FUNCTION_BLOCK FB_FBD_IL_LD_SamplePOU
VAR_INPUT
//	eOperation	: INT;
	eOperation	: E_Operation;
END_VAR
VAR_OUTPUT
	iResultC	: DINT;
END_VAR
VAR
	arrDataA	: ARRAY [1..iMax] OF DINT;
	arrDataB	: ARRAY [1..iMax] OF DINT;
	arrDataC	: ARRAY [1..iMax] OF DINT;
	I 			: DINT;
	bInit		: BOOL := TRUE;
	bEnd		: BOOL;
	bRepeat		: BOOL;
	bAtTheEnd	: BOOL;
END_VAR
VAR CONSTANT
	iMax 		: DINT := 10;
END_VAR
VAR // added by the converter: edge detectors and wires of the graphical bodies
    _w1, _w2, _w3, _w4, _w5, _w6, _w7 : DINT;
END_VAR

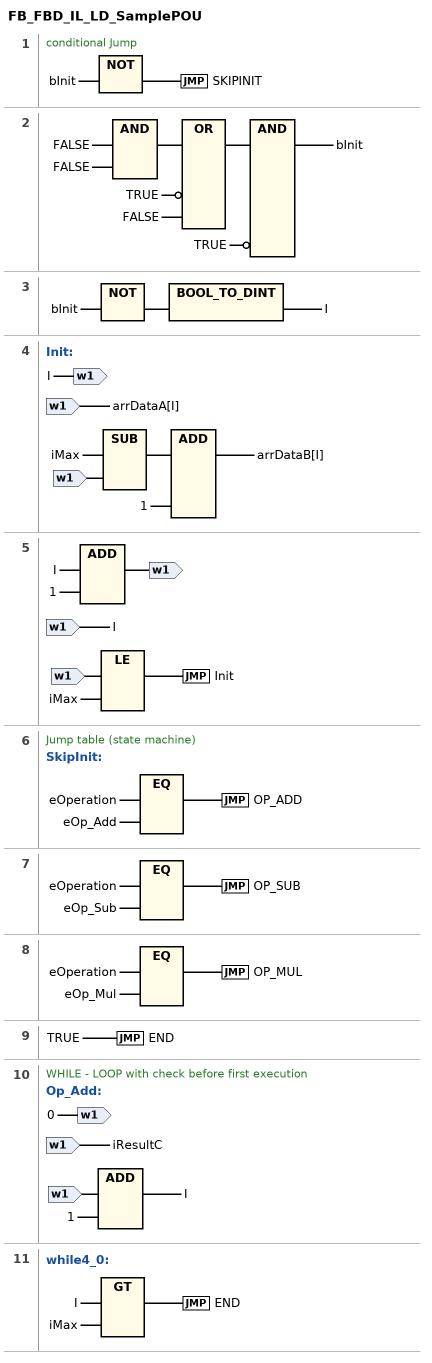
// NETWORK 1
//  conditional Jump
IF NOT bInit THEN JMP SKIPINIT; END_IF

// NETWORK 2
bInit := (FALSE AND FALSE OR NOT TRUE OR FALSE) AND NOT TRUE;

// NETWORK 3
I := BOOL_TO_DINT(NOT bInit);

// NETWORK 4
Init:
arrDataA[I] := I;
arrDataB[I] := (iMax - I) + 1;

// NETWORK 5
_w1 := I + 1;
I := _w1;
IF _w1 <= iMax THEN JMP Init; END_IF

// NETWORK 6
//  Jump table (state machine)
SkipInit:
IF eOperation = eOp_Add THEN JMP OP_ADD; END_IF

// NETWORK 7
IF eOperation = eOp_Sub THEN JMP OP_SUB; END_IF

// NETWORK 8
IF eOperation = eOp_Mul THEN JMP OP_MUL; END_IF

// NETWORK 9
JMP END;

// NETWORK 10
//  WHILE - LOOP with check before first execution
Op_Add:
iResultC := 0;
I := 0 + 1;

// NETWORK 11
while4_0:
IF I > iMax THEN JMP END; END_IF

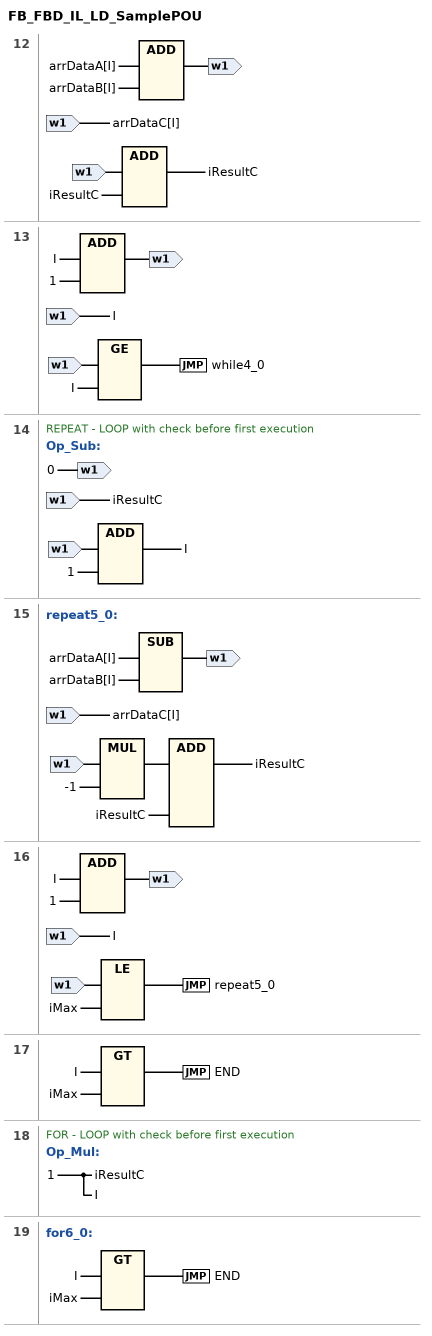
// NETWORK 12
_w2 := arrDataA[I] + arrDataB[I];
arrDataC[I] := _w2;
iResultC := _w2 + iResultC;

// NETWORK 13
_w3 := I + 1;
I := _w3;
IF _w3 >= I THEN JMP while4_0; END_IF

// NETWORK 14
//  REPEAT - LOOP with check before first execution
Op_Sub:
iResultC := 0;
I := 0 + 1;

// NETWORK 15
repeat5_0:
_w4 := arrDataA[I] - arrDataB[I];
arrDataC[I] := _w4;
iResultC := _w4 * -1 + iResultC;

// NETWORK 16
_w5 := I + 1;
I := _w5;
IF _w5 <= iMax THEN JMP repeat5_0; END_IF

// NETWORK 17
IF I > iMax THEN JMP END; END_IF

// NETWORK 18
//  FOR - LOOP with check before first execution
Op_Mul:
iResultC := 1;
I := 1;

// NETWORK 19
for6_0:
IF I > iMax THEN JMP END; END_IF

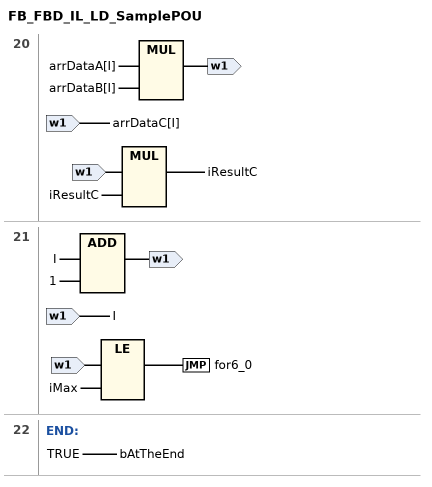
// NETWORK 20
_w6 := arrDataA[I] * arrDataB[I];
arrDataC[I] := _w6;
iResultC := _w6 * iResultC;

// NETWORK 21
_w7 := I + 1;
I := _w7;
IF _w7 <= iMax THEN JMP for6_0; END_IF

// NETWORK 22
END:
bAtTheEnd := TRUE;

END_FUNCTION_BLOCK

(* stored: Version 1.1.0.1, ProductVersion 3.1.4024.11
   POU FB_FBD_IL_LD_SamplePOU: Id {ef69e7da-122c-43e1-906c-30c0cfcbbd23}, SpecialFunc None *)
